// TwinCAT 3 PLC project Library
// libraries:
//   Tc2_Standard, * (Beckhoff Automation GmbH)
// project tree:
//   / FB_Filter.TcPOU, E_State.TcDUT

// ---- E_State.TcDUT

// :Description: Filter state (library copy).
TYPE E_State :
(
    Idle := 0,
    Running := 1,
    Errored := 2
);
END_TYPE

// ---- FB_Filter.TcPOU

// :Description: Rolling-average filter (library code under test).
FUNCTION_BLOCK FB_Filter
VAR_INPUT
    input : LREAL;
END_VAR
VAR_OUTPUT
    output : LREAL;
END_VAR
VAR
    state : E_State := E_State.Idle;
END_VAR


output := input;


// :Description: Advance the filter by one sample.
METHOD Step : LREAL
VAR_INPUT
    sample : LREAL;
END_VAR

Step := sample;
END_METHOD

END_FUNCTION_BLOCK
